FUNCTION_BLOCK CellSensor
VAR
	OKtoRelase 	: BOOL;
	Feeded	: BOOL;
	
END_VAR

METHOD mFeeded : BOOL
VAR_INPUT
END_VAR
Feeded := True;
END_METHOD

METHOD mOKtoRelase : BOOL
VAR_INPUT
END_VAR
OKtoRelase := TRUE;
END_METHOD

PROPERTY pFeeded : BOOL
GET
pFeeded := Feeded;
END_GET
SET
Feeded := pFeeded;
END_SET
END_PROPERTY

PROPERTY pOKtoRelase : BOOL
GET
pOKtoRelase := OKtoRelase;
END_GET
SET
OKtoRelase := pOKtoRelase;
END_SET
END_PROPERTY

END_FUNCTION_BLOCK

(* stored: Version 1.1.0.1, ProductVersion 3.1.4024.9
   POU CellSensor: Id {0062affa-878e-4430-a5f0-cece8346cff4}, SpecialFunc None
   Method mFeeded: Id {a9346240-3726-4ae6-952d-d4b3065614cd}
   Method mOKtoRelase: Id {39654db2-bdff-4174-b61f-9e0c3fcfc6fc}
   Property pFeeded: Id {b4daa3ea-3b61-4054-9030-982b4c281dfc}
   Get Get: Id {556c5342-2af1-48da-b195-15f4bf830677}
   Set Set: Id {0feb8faf-8ff2-4a65-89f9-841faacdd8c2}
   Property pOKtoRelase: Id {4c97c793-9697-4f25-948d-3698a5eea168}
   Get Get: Id {fdc7d8eb-4599-4d01-85d6-0bac86ee6990}
   Set Set: Id {9d1eac1e-f659-44c7-befa-44ab1bac9b3d} *)
